// TIA Portal V20 export
FUNCTION_BLOCK "Q_DAS"   // FB75, LAD
// stored: Access Published, MemoryReserve 100, Namespace Unit1, SetENOAutomatically false
   VAR
      m1 : Bool;
   END_VAR
BEGIN

REGION Network 1
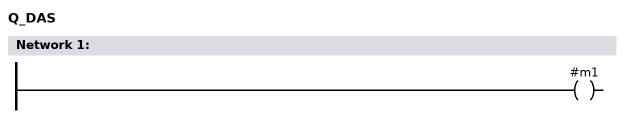
   RUNG wire#powerrail
      Coil( #m1 )
   END_RUNG
   // the same network as SCL:
   #m1 := TRUE;
END_REGION
END_FUNCTION_BLOCK
